FUNCTION_BLOCK FB_Beckhoff_EL6001_Test EXTENDS TcUnit.FB_TestSuite
VAR
	_fbDevice 	: FB_Beckhoff_EL6001;
	_nExpected 	: UINT;
	_nResult 	: UINT;
END_VAR

TestProperties();
TestState();

METHOD TestProperties : REFERENCE TO FB_Test
VAR
	bExpected 		: BOOL;
	bResult 		: BOOL;
END_VAR
TEST('TransmitRequest FALSE');
bExpected := FALSE; 
_fbDevice();
_fbDevice.Control := 0;
_fbDevice();
bResult := _fbDevice.TransmitRequest;
AssertEquals(Expected := bExpected,
             Actual := bResult,
             Message := 'TransmitRequest value is not correct');		
TEST_FINISHED();

TEST('TransmitRequest TRUE');
bExpected := TRUE; 
_fbDevice();
_fbDevice.Control := 1;
_fbDevice();
bResult := _fbDevice.TransmitRequest;
AssertEquals(Expected := bExpected,
             Actual := bResult,
             Message := 'TransmitRequest value is not correct');		
TEST_FINISHED();

TEST('ReceiveAccepted FALSE');
bExpected := FALSE; 
_fbDevice();
_fbDevice.Control := 0;
_fbDevice();
bResult := _fbDevice.ReceiveAccepted;
AssertEquals(Expected := bExpected,
             Actual := bResult,
             Message := 'ReceiveAccepted value is not correct');		
TEST_FINISHED();

TEST('ReceiveAccepted TRUE');
bExpected := TRUE; 
_fbDevice();
_fbDevice.Control := 2;
_fbDevice();
bResult := _fbDevice.ReceiveAccepted;
AssertEquals(Expected := bExpected,
             Actual := bResult,
             Message := 'ReceiveAccepted value is not correct');		
TEST_FINISHED();

TEST('InitRequest TRUE');
bExpected := TRUE; 
_fbDevice();
_fbDevice.Control := 4;
_fbDevice();
bResult := _fbDevice.InitRequest;
AssertEquals(Expected := bExpected,
             Actual := bResult,
             Message := 'InitRequest value is not correct');		
TEST_FINISHED();

TEST('SendContinuous TRUE');
bExpected := TRUE; 
_fbDevice.Control := 0;
_fbDevice();
_fbDevice.Control := 9;
_fbDevice();
bResult := _fbDevice.SendContinuous;
AssertEquals(Expected := bExpected,
             Actual := bResult,
             Message := 'SendContinuous value is not correct');		
TEST_FINISHED();
END_METHOD

METHOD TestState : REFERENCE TO FB_Test
VAR
	bResult 		: BOOL;
	nDataSend 		:  ARRAY[0..50] OF BYTE;
END_VAR
TEST('Transition: INIT - READY');
_fbDevice.Control := 0;
_fbDevice.State := E_Beckhoff_EL6001_State.INIT;	
_fbDevice();

AssertTRUE(_fbDevice.State = E_Beckhoff_EL6001_State.READY, 'State value is not correct');
	
TEST_FINISHED();

TEST('Transition: READY - TRANSMIT');
_fbDevice.Control := 0;
_fbDevice.State := E_Beckhoff_EL6001_State.READY;	
_fbDevice();

_fbDevice.Control := 257;
_fbDevice();

AssertTRUE(_fbDevice.State = E_Beckhoff_EL6001_State.TRANSMIT, 'State value is not correct');
	
TEST_FINISHED();

TEST('Transition: READY - RECEIVE');
_fbDevice.Control := 0;
_fbDevice.State := E_Beckhoff_EL6001_State.READY;	
_fbDevice();

_fbDevice.bSend := TRUE;
_fbDevice.pDataIn := ADR(nDataSend);
_fbDevice.nLength := 1;
_fbDevice.Control := 1;
_fbDevice();

_fbDevice.bSend := FALSE;
_fbDevice.nLength := 0;

AssertTRUE(_fbDevice.State = E_Beckhoff_EL6001_State.RECEIVE, 'State value is not correct');
TEST_FINISHED();
END_METHOD

END_FUNCTION_BLOCK

(* stored: Version 1.1.0.1, ProductVersion 3.1.4024.12
   POU FB_Beckhoff_EL6001_Test: Id {6ec7a068-08cf-0312-2173-c65c8073149f}, SpecialFunc None
   Method TestProperties: Id {b3008bee-f5e3-0c99-3758-dd76255e7318}
   Method TestState: Id {4b7115e8-c51d-08ad-0d86-56821691d517} *)
